{attribute 'qualified_only'}
{attribute 'strict'}
{attribute 'to_string'}
TYPE ST160_CETA_e :
(
    RESET := 0, // Reset

    INIT := 100, // Initialisieren 
    Init_pneumatics,
    Init_vertical_down,

    READY := 999,  // READY to Start, Init Done 
    START := 1000, // Start Zyklisch
    MOVER_FREE_OP, // Ab here, operation without mover can be done

    waitOnMover,     // wait until the mover is there
    MOVER_NEEDED_OP, // Since here, a mover in position is needed to perform the action

    handling_down, // 
    vertical_up,   // 
    seal_piece,   //
    CETA_start,    // 
    CETA_wait_on_result, // 
    CETA_read,     // 
    unseal_piece,   //
    vertical_down, // 
    handling_up,   // 

    SYNC_MOVER_LEAVE, // MoverMan need to take the mover
    DONE := 8000,     // Ablauf beendet 
    ERROR := 9000,    // Fehler 
    _max
);
END_TYPE

(* stored: Version 1.1.0.1, ProductVersion 3.1.4024.6
   EnumerationTextList ST160_CETA_e: Id {f2fd08ad-15a9-43ff-8fb0-c1745a8da171} *)
